SYSTEM RMT_DEV_TEST_INT (* RMT_DEV Test with FB_ADD_INT and E_CTU *)
  (* Standard: 61499-1; Classification: Test; Type: SNAP Test *)
  (* Version 0.2, 2007-11-08, JHC, Holobloc Inc, Removed Applications - not interesting. *)
  (* Version 0.1, 2005-05-17, JHC, Rockwell Automation, Changed sockets 1025-6 to 1031-2 for WXP compatibility. *)
  (* Version 0.0, 2003-07-12, JHC, Rockwell Automation, Modified from RMT_DEV_TEST. *)
  DEVICE DEV_TESTER : FRAME_DEVICE(BOUNDS := [50,50,190,250], GRID := [2,1])
    RESOURCE RES1 : PANEL_RESOURCE
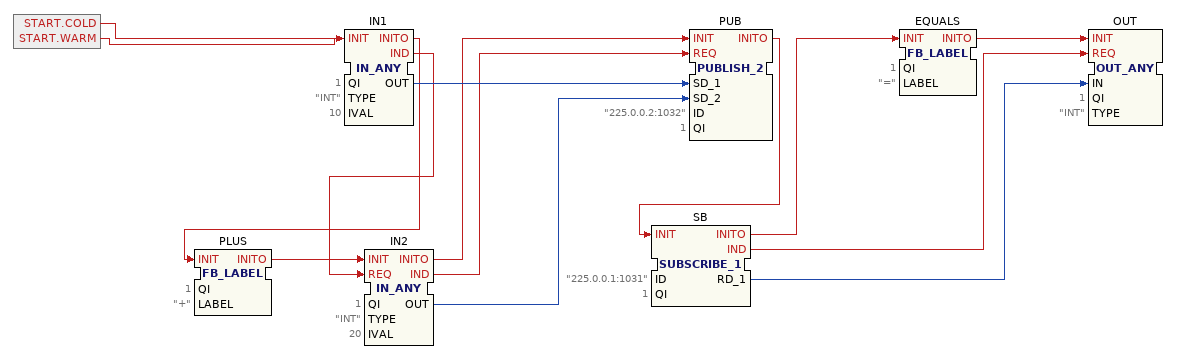
      FBS
        IN1 : IN_ANY(QI := 1, TYPE := "INT", IVAL := 10);
        PLUS : FB_LABEL(QI := 1, LABEL := "+");
        IN2 : IN_ANY(QI := 1, TYPE := "INT", IVAL := 20);
        PUB : PUBLISH_2(ID := "225.0.0.2:1032", QI := 1);
        SB : SUBSCRIBE_1(ID := "225.0.0.1:1031", QI := 1);
        EQUALS : FB_LABEL(QI := 1, LABEL := "=");
        OUT : OUT_ANY(QI := 1, TYPE := "INT");
      END_FBS
      EVENT_CONNECTIONS
        START.COLD TO IN1.INIT;
        START.WARM TO IN1.INIT;
        IN1.INITO TO PLUS.INIT;
        PLUS.INITO TO IN2.INIT;
        IN2.INITO TO PUB.INIT;
        PUB.INITO TO SB.INIT;
        SB.INITO TO EQUALS.INIT;
        EQUALS.INITO TO OUT.INIT;
        IN1.IND TO IN2.REQ;
        IN2.IND TO PUB.REQ;
        SB.IND TO OUT.REQ;
      END_CONNECTIONS
      DATA_CONNECTIONS
        IN1.OUT TO PUB.SD_1;
        IN2.OUT TO PUB.SD_2;
        SB.RD_1 TO OUT.IN;
      END_CONNECTIONS
    END_RESOURCE
    RESOURCE RES2 : PANEL_RESOURCE
      FBS
        RUNSTOP : RADIO_BOOL(QI := 1, LABEL0 := "STOP", LABEL1 := "RUN");
        RESET : IN_EVENT(QI := 1, LABEL := "RESET");
        PUB0 : PUBLISH_0(QI := 1, ID := "225.0.0.5:1029");
        PV : IN_ANY(QI := 1, IVAL := 10, TYPE := "UINT");
        PV_LBL : FB_LABEL(QI := 1, LABEL := "PV");
        DT : IN_ANY(QI := 1, TYPE := "TIME", IVAL := t#500ms);
        DT_LBL : FB_LABEL(QI := 1, LABEL := "DT");
        PUB : PUBLISH_3(QI := 1, ID := "225.0.0.3:1027");
        SB : SUBSCRIBE_2(QI := 1, ID := "225.0.0.4:1028");
        Q : OUT_BOOL(QI := 1, LABEL := "Q", C0 := COLOR#red, C1 := COLOR#green);
        CV : OUT_ANY(QI := 1, TYPE := "UINT");
      END_FBS
      EVENT_CONNECTIONS
        START.COLD TO RUNSTOP.INIT;
        START.WARM TO RUNSTOP.INIT;
        RUNSTOP.INITO TO RESET.INIT;
        RESET.INITO TO PUB0.INIT;
        PUB0.INITO TO PV.INIT;
        PV.INITO TO PV_LBL.INIT;
        PV_LBL.INITO TO DT.INIT;
        DT.INITO TO DT_LBL.INIT;
        DT_LBL.INITO TO PUB.INIT;
        PUB.INITO TO SB.INIT;
        SB.INITO TO CV.INIT;
        CV.INITO TO Q.INIT;
        RUNSTOP.CNF TO PV.REQ;
        RUNSTOP.IND TO PV.REQ;
        RESET.IND TO PUB0.REQ;
        PV.IND TO DT.REQ;
        DT.IND TO PUB.REQ;
        SB.IND TO Q.REQ;
        Q.CNF TO CV.REQ;
      END_CONNECTIONS
      DATA_CONNECTIONS
        RUNSTOP.OUT TO PUB.SD_1;
        PV.OUT TO PUB.SD_3;
        DT.OUT TO PUB.SD_2;
        SB.RD_1 TO Q.IN;
        SB.RD_2 TO CV.IN;
      END_CONNECTIONS
    END_RESOURCE
  END_DEVICE
  DEVICE DEV1 : RMT_DEV(MGR_ID := "192.168.1.5:61499")
    RESOURCE RES1 : EMB_RES
      FBS
        FF : E_SR;
        SB : SUBSCRIBE_2(ID := "225.0.0.2:1032");
        AD : FB_ADD_INT;
        PUB : PUBLISH_1(ID := "225.0.0.1:1031");
      END_FBS
      EVENT_CONNECTIONS
        START.COLD TO FF.S;
        START.WARM TO FF.S;
        START.STOP TO FF.R;
        FF.EO TO SB.INIT;
        SB.INITO TO PUB.INIT;
        SB.IND TO AD.REQ;
        AD.CNF TO PUB.REQ;
      END_CONNECTIONS
      DATA_CONNECTIONS
        SB.RD_1 TO AD.IN1;
        SB.RD_2 TO AD.IN2;
        AD.OUT TO PUB.SD_1;
        FF.Q TO SB.QI;
        SB.QO TO PUB.QI;
      END_CONNECTIONS
    END_RESOURCE
    RESOURCE RES2 : EMB_RES
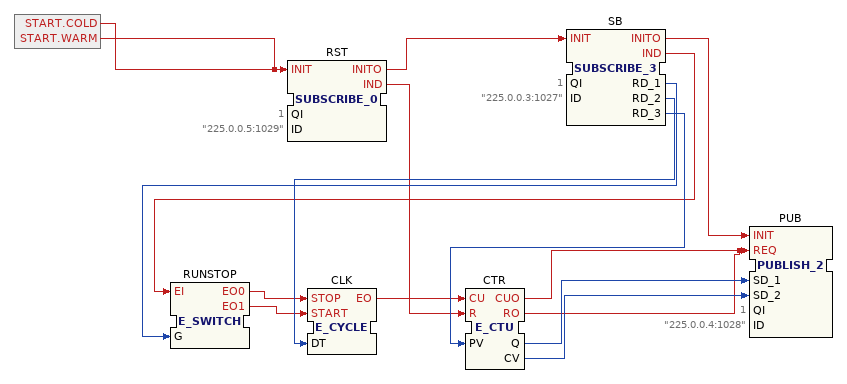
      FBS
        SB : SUBSCRIBE_3(QI := 1, ID := "225.0.0.3:1027");
        RST : SUBSCRIBE_0(QI := 1, ID := "225.0.0.5:1029");
        RUNSTOP : E_SWITCH;
        CLK : E_CYCLE;
        CTR : E_CTU;
        PUB : PUBLISH_2(QI := 1, ID := "225.0.0.4:1028");
      END_FBS
      EVENT_CONNECTIONS
        START.COLD TO RST.INIT;
        START.WARM TO RST.INIT;
        RST.INITO TO SB.INIT;
        SB.INITO TO PUB.INIT;
        SB.IND TO RUNSTOP.EI;
        RUNSTOP.EO0 TO CLK.STOP;
        RUNSTOP.EO1 TO CLK.START;
        CLK.EO TO CTR.CU;
        RST.IND TO CTR.R;
        CTR.CUO TO PUB.REQ;
        CTR.RO TO PUB.REQ;
      END_CONNECTIONS
      DATA_CONNECTIONS
        SB.RD_1 TO RUNSTOP.G;
        SB.RD_2 TO CLK.DT;
        SB.RD_3 TO CTR.PV;
        CTR.Q TO PUB.SD_1;
        CTR.CV TO PUB.SD_2;
      END_CONNECTIONS
    END_RESOURCE
    RESOURCE MGR : RMT_RES
    END_RESOURCE
  END_DEVICE
END_SYSTEM
